FUNCTION_BLOCK Woltz_Object EXTENDS Person_Object
VAR
    _Khartoum : Horse_Object(THIS^);
END_VAR

METHOD ThinkCarefully
IF _Khartoum._isAlive THEN
    _refuseFavor := TRUE;
    _grantFavor := FALSE;
ELSE
    _refuseFavor := FALSE;
    _grantFavor := TRUE;
END_IF;
END_METHOD

END_FUNCTION_BLOCK

(* stored: Version 1.1.0.1, ProductVersion 3.1.4024.9
   POU Woltz_Object: Id {5f3c91dc-f440-03e0-2cf3-ff1d155e00ef}, SpecialFunc None
   Method ThinkCarefully: Id {8b60946d-07cc-0160-2d88-fa7c8575d7b9} *)
